// TIA Portal V21 export
VAR_GLOBAL   // PLC tag table "KAllValv"
END_VAR
VAR_GLOBAL CONSTANT   // user constants
   KAllValv_TimeOutPosiz : Int := 1;
   KAllValv_ValvolaNonInAuto : Int := 2;
   KAllValv_ResetRichiesto : Int := 3;
   KAllValv_ByPassFinecorsa : Int := 4;
END_VAR
